// TIA Portal V20 export
TYPE "LKinCtrl_typeCOffCmdInInternal"
   STRUCT
      cmdType : Int := -1;   // 1: MoveLinAbs; 2: MoveLinRel; 3: MoveCircAbs; 4: MoveCircRel; 5: MoveDirectAbs; 6: MoveDirectRel; 10: TrackConveyorBelt; 100: WaitTime; 40/41/42: ContourOffset; 0: FlagOnlyCmd; -1: End of List
      endPoint : "LKinCtrl_typeCOff3DPoint";   // End point of command
      circleMode : DInt;   // 0: auxPoint defines point on circle line; 1: auxPoint defines circle center; 2: radius and endPoint define circle segment
      circleCenterPoint : "LKinCtrl_typeCOff3DPoint";   // Center point of circle
      circleIntermediatePoint : "LKinCtrl_typeCOff3DPoint";   // Intermediate point of circle
      circleRadius : LReal;   // Radius of circle
      circleAngle : LReal;   // Angle of circle
      pathChoice : DInt;   // circMode(0): not relevant; circMode(1): 0: pos direction; 1: neg direction; circMode(2): 0: short pos segment; 1: short neg segment; 2: long pos segment; 3: long neg segment
      circlePlane : DInt;   // circMode(0): not relevant; circMode(1+2): 0: XZ; 1: YZ; 2: XY
      transitionParameter1 : LReal;   // Transition parameter
      bufferMode : DInt;   // 1: standstill between commands, 2: blending with lower speed; 5: blending with higher speed
   END_STRUCT;
END_TYPE
